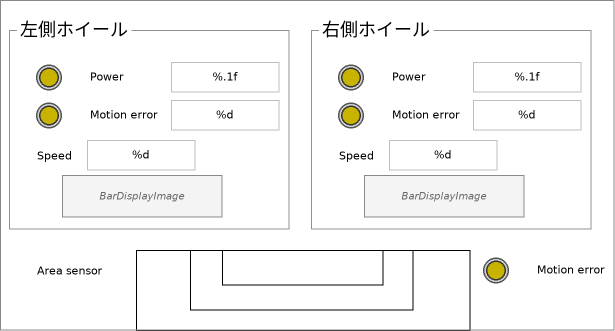
VISUALIZATION main  // 615x331
    GroupBox (9,22 280x207), "左側ホイール"
        BarDisplayImage (53,153 160x42), value: MAIN.diSpeed, style: BarDisplayImage-Gray, scale format: %.1f, scale 0..100
        Lamp1 (25,40 30x31), variable: MAIN.stAxis[1].Status.MotionState > 1, style: Lamp-Lamp1-Yellow
        Label (78,40 81x30), "Power"
        Lamp1 (25,78 30x31), variable: MAIN.stAxis[1].Status.Error, style: Lamp-Lamp1-Yellow
        Textfield (78,118 108x30), "%d", text variable: MAIN.lrVelocity
        Textfield (162,40 108x30), "%.1f", text variable: MAIN.lrOverride
        Label (25,119 47x30), "Speed"
    Label (87,100 81x30), "Motion error"
    Textfield (171,100 108x30), "%d", text variable: MAIN.stAxis[1].Status.ErrorID
    GroupBox (311,22 280x207), "右側ホイール"
        BarDisplayImage (53,153 160x42), value: MAIN.diSpeed, style: BarDisplayImage-Gray, scale format: %.1f, scale 0..100
        Lamp1 (25,40 30x31), variable: MAIN.stAxis[2].Status.MotionState > 1, style: Lamp-Lamp1-Yellow
        Label (78,40 81x30), "Power"
        Lamp1 (25,78 30x31), variable: MAIN.stAxis[2].Status.Error, style: Lamp-Lamp1-Yellow
        Textfield (78,118 108x30), "%d", text variable: MAIN.lrVelocity
        Textfield (162,40 108x30), "%.1f", text variable: MAIN.lrOverride
        Label (25,119 47x30), "Speed"
    Label (389,100 81x30), "Motion error"
    Textfield (473,100 108x30), "%d", text variable: MAIN.stAxis[2].Status.ErrorID
    RoundedRectangle (136,250 334x81), colour toggle: MAIN.bWarningSigna0l
    RoundedRectangle (190,250 223x60), colour toggle: MAIN.bWarningSigna02
    RoundedRectangle (222,250 161x35), colour toggle: MAIN.Mode=AreaStatus.Hazard
    Label (534,255 81x30), "Motion error"
    Lamp1 (481,255 30x31), variable: MAIN.bSafetyRun, style: Lamp-Lamp1-Yellow
    Label (34,256 81x30), "Area sensor"
END_VISUALIZATION

(* stored: Version 1.1.0.1
   Visu main: Id {1c31de08-d59a-40c7-a17e-5827b96208d1} *)
